// TIA Portal project "BHX_PLC_2_V17" (V17)

(* hardware
DEVICE "ET 200SP station_1"  ET 200SP-Station
   slot 0: "Rack_0"  Rack  6ES5 710-8MAx1
   slot 1: "k1bhx01cpu"  CPU 1510SP-1 PN  6ES7 510-1DJ01-0AB0  V2.8
      slot 32768: "PROFINET interface_1"  X1
         slot 32771: "Port_3"  X1 P3
   slot 2: "DI 8x24VDC BA_1"  DI 8x24VDC BA  6ES7 131-6BF01-0AA0  V0.0
      slot 1: "DI 8x24VDC BA_1"  DI 8x24VDC BA
   slot 3: "DI 8x24VDC BA_2"  DI 8x24VDC BA  6ES7 131-6BF01-0AA0  V0.0
      slot 1: "DI 8x24VDC BA_2"  DI 8x24VDC BA
   slot 4: "DQ 8x24VDC/0.5A ST_1"  DQ 8x24VDC/0.5A ST  6ES7 132-6BF01-0BA0  V0.0
      slot 1: "DQ 8x24VDC/0.5A ST_1"  DQ 8x24VDC/0.5A ST
   slot 5: "Server module_1"  Server module  6ES7 193-6PA00-0AA0  V1.1
      slot 1: "Server module_1"  Server module
   slot 127: "BA 2xRJ45"  BA 2xRJ45  6ES7 193-6AR00-0AA0  V0.0
      slot 32769: "Port_1"  X1 P1  6ES7 193-6AR00-0AA0
      slot 32770: "Port_2"  X1 P2  6ES7 193-6AR00-0AA0
DEVICE "ET 200SP station_2"  ET 200SP-Station
   slot 0: "Rack_0"  Rack  6ES5 710-8MAx1
   slot 0: "et-bhx"  IM 155-6 PN ST  6ES7 155-6AU01-0BN0  V4.1
   slot 1: "DI 8x24VDC BA_1"  DI 8x24VDC BA  6ES7 131-6BF01-0AA0  V0.0
      slot 1: "DI 8x24VDC BA_1"  DI 8x24VDC BA
   slot 2: "DQ 8x24VDC/0.5A ST_1"  DQ 8x24VDC/0.5A ST  6ES7 132-6BF01-0BA0  V0.0
      slot 1: "DQ 8x24VDC/0.5A ST_1"  DQ 8x24VDC/0.5A ST
   slot 3: "AI 4xU/I 2-wire ST_1"  AI 4xU/I 2-wire ST  6ES7 134-6HD01-0BA1  V2.0
      slot 1: "AI 4xU/I 2-wire ST_1"  AI 4xU/I 2-wire ST
   slot 4: "Server module_1"  Server module  6ES7 193-6PA00-0AA0  V1.1
      slot 1: "Server module_1"  Server module
   slot 127: "BA 2xRJ45"  BA 2xRJ45  6ES7 193-6AR00-0AA0  V0.0
      slot 1: "Port_1"  X1 P1 R  6ES7 193-6AR00-0AA0  V0.0
      slot 2: "Port_2"  X1 P2 R  6ES7 193-6AR00-0AA0  V0.0
DEVICE "GSD device_1"  GSD.Device.PN
   slot 0: "Rack"  Rack  V1.0
   slot 0: "k1bhx011"  KRC4-ProfiNet_4.1  0x300  V4.1
      slot 0: "KRC4-ProfiNet_4.1"  KRC4-ProfiNet_4.1
      slot 1: "Interface1"  Interface1
         slot 1: "Port1"  Port1
   slot 2: "1024 digital in- and outputs_1"  1024 digital in- and outputs  KUKA Device IO1024
      slot 0: "1024 digital in- and outputs"  1024 digital in- and outputs
DEVICE "GSD device_2"  GSD.Device.PN
   slot 0: "Rack"  Rack  V1.0
   slot 0: "matrixbhx"  Matrix 320  M320  V1.37.0
      slot 0: "Matrix 320"  Matrix 320
      slot 1: "1 Port PN-RT"  1 Port PN-RT
         slot 1: "Port 1"  Port 1
   slot 1: "Virtual 8 Byte Output"  Virtual 8 Byte Output
      slot 0: "Virtual 8 Byte Output"  Virtual 8 Byte Output
   slot 2: "Virtual 64 Byte Input"  Virtual 64 Byte Input
      slot 0: "Virtual 64 Byte Input"  Virtual 64 Byte Input
*)

// ===== PLC "k1bhx01cpu"  CPU 1510SP-1 PN =====

VAR_GLOBAL   // PLC tag table "PLC_Machine_IO"
   "PLC_WorkpieceAtStopper" AT %Q0.0 : Bool;
   "PLC_InfeedAreaFree" AT %Q0.1 : Bool;
   "PLC_OutfeedAreaFree" AT %Q0.2 : Bool;
   "PLC_OpenClamps" AT %Q0.3 : Bool;
   "PLC_ResetMcc" AT %Q0.4 : Bool;
   "PLC_InfeedPositionFree" AT %I0.0 : Bool;
   "PLC_WorkpieceClamped" AT %I0.1 : Bool;
   "PLC_WorkpieceRdyToTurn" AT %I0.2 : Bool;
   "PLC_WorkpiecePickupPos1" AT %I0.3 : Bool;
   "PLC_WorkpiecePickupPos2" AT %I0.4 : Bool;
   "PLC_AutoFeedingModeActive" AT %I0.5 : Bool;
   "PLC_StopperWorkpos" AT %I0.6 : Bool;
END_VAR

VAR_GLOBAL   // PLC tag table "Robot_Machine_IO"
   "WorkpieceAtStopper" AT %I20.0 : Bool;
   "InfeedAreaFree" AT %I20.1 : Bool;
   "OutfeedAreaFree" AT %I20.2 : Bool;
   "OpenClamps" AT %I20.3 : Bool;
   "ResetMcc" AT %I20.4 : Bool;
   "InfeedPositionFree" AT %Q20.0 : Bool;
   "WorkpieceClamped" AT %Q20.1 : Bool;
   "WorkpieceRdyToTurn" AT %Q20.2 : Bool;
   "WorkpiecePickupPos1" AT %Q20.3 : Bool;
   "WorkpiecePickupPos2" AT %Q20.4 : Bool;
   "AutoFeedingModeActive" AT %Q20.5 : Bool;
   "StopperWorkpos" AT %Q20.6 : Bool;
END_VAR

VAR_GLOBAL   // PLC tag table "ET200_Gripper"
   "InGripperMainHome1" AT %I10.0 : Bool;
   "InGripperRetracted" AT %I10.1 : Bool;
   "InGripperMainHome2" AT %I10.2 : Bool;
   "InGripperFeederHome" AT %I10.3 : Bool;
   "OutVacuumON" AT %Q10.0 : Bool;
   "InGripperGerconNC" AT %I10.4 : Bool;
   "InGripperVacuumNC" AT %I10.5 : Bool;
   "InGripperRangefinder" AT %IW14 : Int;
   "OutPressureOFF" AT %Q10.1 : Bool;
   "OutGripperMainRetract" AT %Q10.2 : Bool;
   "OutFlow2Part" AT %Q10.3 : Bool;
END_VAR

VAR_GLOBAL   // PLC tag table "KUKA_To_PLC"
   "From_KUKA_ALARM_STOP_KRC" AT %I35.1 : Bool;   // KUKA. Аварийный СТОП (122)
   "From_KUKA_EXT_ACTIVE" AT %I35.7 : Bool;   // KUKA. В режиме Внешняя Автоматика (128)
   "From_KUKA_PERI_RDY_KRC" AT %I35.5 : Bool;   // KUKA. Готовность приводов (126)
   "From_KUKA_STOPMESS_KRC" AT %I35.3 : Bool;   // KUKA. СТОП (124)
   "From_KUKA_IN_HOME_KRC" AT %I36.0 : Bool;   // KUKA. В домашней позиции (129)
   "From_KUKA_PRO_MOVE_KRC" AT %I36.7 : Bool;   // KUKA. Робот в движении (136)
   "From_KUKA_PGNO_REFL_KRC" AT %IW37 : UInt;   // KUKA. Активный номер программы (137-152)
   "From_KUKA_PGNO_REQ_KRC" AT %I36.2 : Bool;   // KUKA. Запрос на новую программу (131)
   "From_KUKA_USER_SAF_KRC" AT %I35.4 : Bool;   // KUKA. Безопасность оператора (125)
   "From_KUKA_ROB_CAL_KRC" AT %I36.1 : Bool;   // KUKA. Юстировка выполнена (130)
   "From_KUKA_I_O_ACTCONF_KRC" AT %I35.2 : Bool;   // KUKA. Внешняя автоматика сконфигурирована (123)
   "From_KUKA_RC_RDY1_KRC" AT %I35.0 : Bool;   // KUKA. Готовность приводов (121)
   "From_KUKA_APPL_RUN_KRC" AT %I36.3 : Bool;   // KUKA. Приложение запущено (132)
   "From_KUKA_Cam" AT %I21.3 : Bool;   // KUKA. Запрос на сканирование (12)
   "From_KUKA_LifeBit" AT %I35.6 : Bool;   // KUKA. Бит Жизни (127)
   "From_KUKA_EXT_FIRST_START" AT %I36.5 : Bool;   // KUKA. Начальный запуск внешней автоматики (134)
   "From_KUKA_SetVacuumON" AT %I21.0 : Bool;   // KUKA. Включить вакуум (9)
   "From_KUKA_SetPressureOFF" AT %I21.1 : Bool;   // KUKA. Выключить давление (10)
   "From_KUKA_SetRetract" AT %I21.2 : Bool;   // KUKA. Задвинуть цилиндры (11)
   "From_KUKA_Flow2PartON" AT %I21.5 : Bool;   // KUKA. Включить поддув деталей (14)
   "From_KUKA_SetFlipClose" AT %I21.4 : Bool;   // KUKA. Закрыть стол переворота(13)
   "From_KUKA_PartOK" AT %I22.0 : Bool;   // KUKA. Деталь ОК (17)
   "From_KUKA_PartMeasuring" AT %I21.7 : Bool;   // KUKA. Измерение детали (16)
   "From_KUKA_PRO_ACT_KRC" AT %I36.6 : Bool;   // KUKA. Программа активна (135)
   "From_KUKA_ERROR_KRC" AT %I36.4 : Bool;   // KUKA. Ошибка на роботе (133)
   "From_KUKA_AXIS_ACT_A1" AT %IW24 : UInt;   // KUKA. Угол поворота оси А1 робота плюс 180 градусов (33-48)
   "From_KUKA_POS_ACT_Z" AT %IW30 : UInt;   // KUKA. Координата Z актуальной позиции робота (81-96)
   "From_KUKA_POS_ACT_Y" AT %IW28 : UInt;   // KUKA. Координата Y актуальной позиции робота (65-80)
   "From_KUKA_POS_ACT_X" AT %IW26 : UInt;   // KUKA. Координата X актуальной позиции робота (49-64)
   "From_KUKA_POS_ACT_A" AT %IW32 : UInt;   // KUKA. Угол A актуальной позиции робота (97-112)
   "From_KUKA_Pallet_Scanned" AT %I39.0 : Bool;   // KUKA. Робот в движении (153)
   "From_KUKA_FlipVacuumOn" AT %I21.6 : Bool;   // KUKA. Включить вакуум стола (15)
   "From_KUKA_Part_Status" AT %IW40 : UInt;   // KUKA. Статус детали (161-176)
   "From_KUKA_Serial_Number" AT %IW42 : UInt;   // KUKA. Серийный номер (177-192)
END_VAR

VAR_GLOBAL   // PLC tag table "PLC_To_KUKA"
   "To_KUKA_Rangefinder" AT %QW43 : UInt;   // PLC. Дальномер (185-200)
   "To_KUKA_Gercon" AT %Q21.4 : Bool;   // PLC. Касание листа нормальное (13)
   "To_KUKA_PLC_STOP" AT %Q32.3 : Bool;   // PLC. ПЛК - СТОП (100)
   "To_KUKA_PAUSE_STOP" AT %Q32.4 : Bool;   // PLC. ПЛК - ПАУЗА (101)
   "To_KUKA_MOVE_ENABLE_KRC" AT %Q35.1 : Bool;   // PLC. Разрешение на перемещение (122)
   "To_KUKA_PGNO_KRC" AT %QW33 : UInt;   // PLC. Номер программы (105-120)
   "To_KUKA_PGNO_VALID_KRC" AT %Q35.6 : Bool;   // PLC. Корректность номера программы 127
   "To_KUKA_PGNO_PARITY" AT %Q35.5 : Bool;   // PLC. Чётность номера программы 126
   "To_KUKA_CONF_MESS" AT %Q35.2 : Bool;   // PLC. Подтверждение сообщения 123
   "To_KUKA_DRIVERS_OFF" AT %Q35.4 : Bool;   // PLC. Отключить привода 125
   "To_KUKA_DRIVERS_ON" AT %Q35.3 : Bool;   // PLC. Включить привода 124
   "To_KUKA_Collision" AT %Q21.5 : Bool;   // PLC. Касание аварийное (14)
   "To_KUKA_QRcode_X" AT %QW37 : UInt;   // PLC. Отклонение по оси X (137-152)
   "To_KUKA_QRcode_Angle" AT %QW41 : UInt;   // PLC. Отклонение по углу (169-184)
   "To_KUKA_EXT_START_KRC" AT %Q35.0 : Bool;   // PLC. Внешний страт (121)
   "To_KUKA_Vacuum_Ok" AT %Q21.6 : Bool;   // PLC. Вакуум ОК (15)
   "To_KUKA_QRcode_Y" AT %QW39 : UInt;   // PLC. Отклонение по оси Y (153-168)
   "To_KUKA_Cam_Ok" AT %Q21.7 : Bool;   // PLC. Камера ОК (16)
   "To_KUKA_IsGripperMainHome" AT %Q21.0 : Bool;   // PLC. Геркон основного цилиндра (9)
   "To_KUKA_IsGripperFeederHome" AT %Q21.1 : Bool;   // PLC. Геркон цилиндра подачи (10)
   "To_KUKA_Part_length_X" AT %QW45 : UInt;   // PLC. Длинна детали по X (201-216)
   "To_KUKA_Part_thickness_Z" AT %QW49 : UInt;   // PLC. Ширина детали по Z (233-248)
   "To_KUKA_GripperRetracted" AT %Q22.0 : Bool;   // PLC. Концевой выключатель (17)
   "To_KUKA_PartEndSwitch_1" AT %Q22.1 : Bool;   // PLC. Концевой выключатель (18)
   "To_KUKA_PartEndSwitch_2" AT %Q22.2 : Bool;   // PLC. Концевой выключатель (19)
   "To_KUKA_Gripper_Sign_X" AT %Q22.3 : Bool;   // PLC. Сдвиг захвата по X (20)
   "To_KUKA_Gripper_Sign_Y" AT %Q22.4 : Bool;   // PLC. Сдвиг захвата по Y (21)
   "To_KUKA_FlipTableOpened" AT %Q22.6 : Bool;   // PLC. Стол для переворота открыт (23)
   "To_KUKA_FlipTableClosed" AT %Q22.7 : Bool;   // PLC. Стол для переворота закрыт (24)
   "To_KUKA_Part_length_Y" AT %QW47 : UInt;   // PLC. Длинна детали по Y (217-232)
   "To_KUKA_QRcode_Z" AT %QW51 : UInt;   // PLC. Отклонение по высоте (249-264)
   "To_KUKA_Part_X" AT %QW53 : UInt;   // PLC. Отклонение по оси X (265-280)
   "To_KUKA_Part_Y" AT %QW55 : UInt;   // PLC. Отклонение по оси Y (281-296)
   "To_KUKA_Part_A" AT %QW59 : UInt;   // PLC. Отклонение по углу (313-328)
   "To_KUKA_Part_Z" AT %QW57 : UInt;   // PLC. Отклонение по высоте (297-312)
   "To_KUKA_Part_Length_X0" AT %QW61 : UInt;   // PLC. Отклонение по высоте (329-344)
   "To_KUKA_Part_Length_Y0" AT %QW63 : UInt;   // PLC. Отклонение по углу (345-360)
   "To_KUKA_Gripper_Within_part" AT %Q22.5 : Bool;   // PLC. Захват соприкасается с деталью полностью (22)
   "To_KUKA_Part_Slot" AT %QW65 : UInt;   // PLC. Отклонение по углу (361-376)
   "To_KUKA_Free_Slot" AT %QW67 : UInt;   // PLC. Отклонение по углу (377-392)
   "To_KUKA_AckPalletScanned" AT %Q32.5 : Bool;   // PLC. Подтверждение сканирования поддона 102
   "To_KUKA_Slot_X" AT %QW69 : UInt;   // PLC. Отклонение по оси X (393-408)
   "To_KUKA_Slot_Y" AT %QW71 : UInt;   // PLC. Отклонение по оси Y (409-424)
   "To_KUKA_Slot_Z" AT %QW73 : UInt;   // PLC. Отклонение по высоте (425-440)
   "To_KUKA_Slot_A" AT %QW75 : UInt;   // PLC. Отклонение по углу (441-456)
   "To_KUKA_WithoutMachine" AT %Q32.6 : Bool;   // PLC. Работа без машины 103
   "To_KUKA_Part_Destination" AT %QW77 : UInt;   // PLC. Назначение детали (457-472)
   "To_KUKA_Out_X" AT %QW79 : UInt;   // PLC. Отклонение по оси X (473-488)
   "To_KUKA_Out_Y" AT %QW81 : UInt;   // PLC. Отклонение по оси Y (489-544)
   "To_KUKA_Out_Z" AT %QW83 : UInt;   // PLC. Отклонение по высоте (505-520)
   "To_KUKA_Out_A" AT %QW85 : UInt;   // PLC. Отклонение по углу (521-536)
END_VAR

VAR_GLOBAL   // PLC tag table "Matrix"
   "MatrixPhase_ON" AT %Q148.7 : Bool;
   "MatrixGoobRead" AT %I148.0 : Bool;
   "MatrixBadRead" AT %I148.1 : Bool;
END_VAR

VAR_GLOBAL   // PLC tag table "Operator_panel"
   "button_Alarm" AT %I1.0 : Bool;
   "button_Pause" AT %I1.1 : Bool;
   "button_Reset" AT %I1.2 : Bool;
   "button_Start" AT %I1.3 : Bool;
END_VAR

VAR_GLOBAL   // PLC tag table "FlipTable"
   "OutFlipClose" AT %Q0.5 : Bool;
   "OutFlipVacuumOn" AT %Q0.6 : Bool;
END_VAR

VAR_GLOBAL   // PLC tag table "RobotTask"
   "task_status" AT %Q1000.0 : "Char_30";
   "part_status" AT %Q1030.0 : "Char_30";
END_VAR

VAR_GLOBAL   // PLC tag table "PLC_To_VC"
   "To_VC_Rangefinder" AT %QW343 : UInt;   // PLC. Дальномер (185-200)
   "To_VC_Gercon" AT %Q321.4 : Bool;   // PLC. Касание листа нормальное (13)
   "To_VC_PLC_STOP" AT %Q332.3 : Bool;   // PLC. ПЛК - СТОП (100)
   "To_VC_PAUSE_STOP" AT %Q332.4 : Bool;   // PLC. ПЛК - ПАУЗА (101)
   "To_VC_MOVE_ENABLE_KRC" AT %Q335.1 : Bool;   // PLC. Разрешение на перемещение (122)
   "To_VC_PGNO_KRC" AT %QW333 : UInt;   // PLC. Номер программы (105-120)
   "To_VC_PGNO_VALID_KRC" AT %Q335.6 : Bool;   // PLC. Корректность номера программы 127
   "To_VC_PGNO_PARITY" AT %Q335.5 : Bool;   // PLC. Чётность номера программы 126
   "To_VC_CONF_MESS" AT %Q335.2 : Bool;   // PLC. Подтверждение сообщения 123
   "To_VC_DRIVERS_OFF" AT %Q335.4 : Bool;   // PLC. Отключить привода 125
   "To_VC_DRIVERS_ON" AT %Q335.3 : Bool;   // PLC. Включить привода 124
   "To_VC_Collision" AT %Q321.5 : Bool;   // PLC. Касание аварийное (14)
   "To_VC_QRcode_X" AT %QW337 : UInt;   // PLC. Отклонение по оси X (137-152)
   "To_VC_QRcode_Angle" AT %QW341 : UInt;   // PLC. Отклонение по углу (169-184)
   "To_VC_EXT_START_KRC" AT %Q335.0 : Bool;   // PLC. Внешний страт (121)
   "To_VC_Vacuum_Ok" AT %Q321.6 : Bool;   // PLC. Вакуум ОК (15)
   "To_VC_QRcode_Y" AT %QW339 : UInt;   // PLC. Отклонение по оси Y (153-168)
   "To_VC_Cam_Ok" AT %Q321.7 : Bool;   // PLC. Камера ОК (16)
   "To_VC_IsGripperMainHome" AT %Q321.0 : Bool;   // PLC. Геркон основного цилиндра (9)
   "To_VC_IsGripperFeederHome" AT %Q321.1 : Bool;   // PLC. Геркон цилиндра подачи (10)
   "To_VC_Part_length_X" AT %QW345 : UInt;   // PLC. Длинна детали по X (201-216)
   "To_VC_Part_thickness_Z" AT %QW349 : UInt;   // PLC. Ширина детали по Z (233-248)
   "To_VC_GripperRetracted" AT %Q322.0 : Bool;   // PLC. Концевой выключатель (17)
   "To_VC_PartEndSwitch_1" AT %Q322.1 : Bool;   // PLC. Концевой выключатель (18)
   "To_VC_PartEndSwitch_2" AT %Q322.2 : Bool;   // PLC. Концевой выключатель (19)
   "To_VC_Gripper_Sign_X" AT %Q322.3 : Bool;   // PLC. Сдвиг захвата по X (20)
   "To_VC_Gripper_Sign_Y" AT %Q322.4 : Bool;   // PLC. Сдвиг захвата по Y (21)
   "To_VC_FlipTableOpened" AT %Q322.6 : Bool;   // PLC. Стол для переворота открыт (23)
   "To_VC_FlipTableClosed" AT %Q322.7 : Bool;   // PLC. Стол для переворота закрыт (24)
   "To_VC_Part_length_Y" AT %QW347 : UInt;   // PLC. Длинна детали по Y (217-232)
   "To_VC_QRcode_Z" AT %QW351 : UInt;   // PLC. Отклонение по высоте (249-264)
   "To_VC_Part_X" AT %QW353 : UInt;   // PLC. Отклонение по оси X (265-280)
   "To_VC_Part_Y" AT %QW355 : UInt;   // PLC. Отклонение по оси Y (281-296)
   "To_VC_Part_A" AT %QW359 : UInt;   // PLC. Отклонение по углу (313-328)
   "To_VC_Part_Z" AT %QW357 : UInt;   // PLC. Отклонение по высоте (297-312)
   "To_VC_Part_Length_X0" AT %QW361 : UInt;   // PLC. Отклонение по высоте (329-344)
   "To_VC_Part_Length_Y0" AT %QW363 : UInt;   // PLC. Отклонение по углу (345-360)
   "To_VC_Gripper_Within_part" AT %Q322.5 : Bool;   // PLC. Захват соприкасается с деталью полностью (22)
   "To_VC_Part_Slot" AT %QW365 : UInt;   // PLC. Отклонение по углу (361-376)
   "To_VC_Free_Slot" AT %QW367 : UInt;   // PLC. Отклонение по углу (377-392)
   "To_VC_AckPalletScanned" AT %Q332.5 : Bool;   // PLC. Подтверждение сканирования поддона 102
   "To_VC_Slot_X" AT %QW369 : UInt;   // PLC. Отклонение по оси X (393-408)
   "To_VC_Slot_Y" AT %QW371 : UInt;   // PLC. Отклонение по оси Y (409-424)
   "To_VC_Slot_Z" AT %QW373 : UInt;   // PLC. Отклонение по высоте (425-440)
   "To_VC_Slot_A" AT %QW375 : UInt;   // PLC. Отклонение по углу (441-456)
   "To_VC_WithoutMachine" AT %Q332.6 : Bool;   // PLC. Работа без машины 103
   "To_VC_Part_Destination" AT %QW377 : UInt;   // PLC. Назначение детали (457-472)
   "To_VC_Out_X" AT %QW379 : UInt;   // PLC. Отклонение по оси X (473-488)
   "To_VC_Out_Y" AT %QW381 : UInt;   // PLC. Отклонение по оси Y (489-544)
   "To_VC_Out_Z" AT %QW383 : UInt;   // PLC. Отклонение по высоте (505-520)
   "To_VC_Out_A" AT %QW385 : UInt;   // PLC. Отклонение по углу (521-536)
   "To_VC_Test_DInt" AT %QD388 : DInt;   // PLC. Tecт
END_VAR

VAR_GLOBAL   // PLC tag table "VC_To_PLC"
   "From_VC_ALARM_STOP_KRC" AT %I335.1 : Bool;   // KUKA. Аварийный СТОП (122)
   "From_VC_EXT_ACTIVE" AT %I335.7 : Bool;   // KUKA. В режиме Внешняя Автоматика (128)
   "From_VC_PERI_RDY_KRC" AT %I335.5 : Bool;   // KUKA. Готовность приводов (126)
   "From_VC_STOPMESS_KRC" AT %I335.3 : Bool;   // KUKA. СТОП (124)
   "From_VC_IN_HOME_KRC" AT %I336.0 : Bool;   // KUKA. В домашней позиции (129)
   "From_VC_PRO_MOVE_KRC" AT %I336.7 : Bool;   // KUKA. Робот в движении (136)
   "From_VC_PGNO_REFL_KRC" AT %IW337 : UInt;   // KUKA. Активный номер программы (137-152)
   "From_VC_PGNO_REQ_KRC" AT %I336.2 : Bool;   // KUKA. Запрос на новую программу (131)
   "From_VC_USER_SAF_KRC" AT %I335.4 : Bool;   // KUKA. Безопасность оператора (125)
   "From_VC_ROB_CAL_KRC" AT %I336.1 : Bool;   // KUKA. Юстировка выполнена (130)
   "From_VC_I_O_ACTCONF_KRC" AT %I335.2 : Bool;   // KUKA. Внешняя автоматика сконфигурирована (123)
   "From_VC_RC_RDY1_KRC" AT %I335.0 : Bool;   // KUKA. Готовность приводов (121)
   "From_VC_APPL_RUN_KRC" AT %I336.3 : Bool;   // KUKA. Приложение запущено (132)
   "From_VC_Cam" AT %I321.3 : Bool;   // KUKA. Запрос на сканирование (12)
   "From_VC_LifeBit" AT %I335.6 : Bool;   // KUKA. Бит Жизни (127)
   "From_VC_EXT_FIRST_START" AT %I336.5 : Bool;   // KUKA. Начальный запуск внешней автоматики (134)
   "From_VC_SetVacuumON" AT %I321.0 : Bool;   // KUKA. Включить вакуум (9)
   "From_VC_SetPressureOFF" AT %I321.1 : Bool;   // KUKA. Выключить давление (10)
   "From_VC_SetRetract" AT %I321.2 : Bool;   // KUKA. Задвинуть цилиндры (11)
   "From_VC_Flow2PartON" AT %I321.5 : Bool;   // KUKA. Включить поддув деталей (14)
   "From_VC_SetFlipClose" AT %I321.4 : Bool;   // KUKA. Закрыть стол переворота(13)
   "From_VC_PartOK" AT %I322.0 : Bool;   // KUKA. Деталь ОК (17)
   "From_VC_PartMeasuring" AT %I321.7 : Bool;   // KUKA. Измерение детали (16)
   "From_VC_PRO_ACT_KRC" AT %I336.6 : Bool;   // KUKA. Программа активна (135)
   "From_VC_ERROR_KRC" AT %I336.4 : Bool;   // KUKA. Ошибка на роботе (133)
   "From_VC_AXIS_ACT_A1" AT %IW324 : UInt;   // KUKA. Угол поворота оси А1 робота плюс 180 градусов (33-48)
   "From_VC_POS_ACT_Z" AT %IW330 : UInt;   // KUKA. Координата Z актуальной позиции робота (81-96)
   "From_VC_POS_ACT_Y" AT %IW328 : UInt;   // KUKA. Координата Y актуальной позиции робота (65-80)
   "From_VC_POS_ACT_X" AT %IW326 : UInt;   // KUKA. Координата X актуальной позиции робота (49-64)
   "From_VC_POS_ACT_A" AT %IW332 : UInt;   // KUKA. Угол A актуальной позиции робота (97-112)
   "From_VC_Pallet_Scanned" AT %I339.0 : Bool;   // KUKA. Робот в движении (153)
   "From_VC_FlipVacuumOn" AT %I321.6 : Bool;   // KUKA. Включить вакуум стола (15)
   "From_VC_Part_Status" AT %IW340 : UInt;   // KUKA. Статус детали (161-176)
   "From_VC_Serial_Number" AT %IW342 : UInt;   // KUKA. Серийный номер (177-192)
END_VAR

TYPE "PLC_Tag"
   STRUCT
      "Name" : String[30];
      "Type" : String[30];
      Use : String[5];
      ReadOnly : USInt;
      DB_number : UInt;
      OffsetByte : UInt;
      OffsetBit : USInt;
      Robot_number : USInt;
   END_STRUCT;
END_TYPE

TYPE "InStatus"
   STRUCT
      previous_programs : Array[1..5] of Int;
      machine_status : String[30];
      robot_status : String[30];
      part_status : String[30];
      operation_types : Array[1..5] of String[30];
      lay_number : Int := -1;
      operation_side : String[4];
      part_side : String[4];
   END_STRUCT;
   // previous_programs[1] := -1;
   // previous_programs[2] := -1;
   // previous_programs[3] := -1;
   // previous_programs[4] := -1;
   // previous_programs[5] := -1;
END_TYPE

TYPE "RobotProgram"
   STRUCT
      trajectory : String[30];
      Entry_Points : Array[1..12] of "EntryPoint";
      OUT_Status : "OutStatus";
   END_STRUCT;
END_TYPE

TYPE "OutStatus"
   STRUCT
      inprocess_task_status : String[30];
      inprocess_part_status : String[30];
      finish_task_status : String[30];
      finish_part_status : String[30];
   END_STRUCT;
END_TYPE

TYPE "EntryPoint"
   STRUCT
      active : Bool;
      previous_trajectory : String[30];
      machine_status : String[30];
      robot_status : String[30];
      part_status : String[30];
      part_destination : String[30];
      operation_type : String[30];
      lay_number : Int := -1;
      operation_side : String[1] := '';
      part_side : String[1] := '';
   END_STRUCT;
END_TYPE

TYPE "TypeRobotTask"
   STRUCT
      not_sended2Arduino : Bool;
      not_sended2BHX : Bool;
      new_part : Bool;
      start_job : Bool;
      reset_job : Bool;
      robot_alarm_reset : Bool;
      "w/o_machine_mode" : Bool;
      gripper_sign_X : Bool;
      gripper_sign_Y : Bool;
      gripper_within_part : Bool;
      robot_pause : Bool;
      pallet_scanned : Bool;
      new_pallet : Bool;
      robot_in_home : Bool;
      program_fullpath : String[99];
      part_length_X : UInt;
      part_length_Y : UInt;
      part_thickness_Z : UInt;
      part_pos_X : Real;
      part_pos_Y : Real;
      part_pos_Z : Real;
      part_angle_A : Real;
      part_side : Char;
      part_slot : USInt;
      free_slot : USInt;
      operation_side : Char;
      operation_number : Int;
      lay_number : Int;
      robot_task_id : LInt;
      robot_id : LInt;
      part_id : LInt;
      part_number : LInt;
      order_id : LInt;
      plc_id : LInt;
      robot_program : UInt;
      operation_type : String[30];
      machine_status : String[30];
      robot_trajectory : String[30];
      robot_status : String[30];
      task_status : String[30];
      part_status : String[30];
      part_source : String[30];
      part_destination : String[30];
      plc_ip : String[30];
      plc_name : String[30];
      robot_name : String[30];
      part_length_X0 : UInt;
      part_length_Y0 : UInt;
      slot_pos_X : Real;
      slot_pos_Y : Real;
      slot_pos_Z : Real;
      slot_angle_A : Real;
      out_pos_X : Real;
      out_pos_Y : Real;
      out_pos_Z : Real;
      out_pos_A : Real;
      robot_serial : UInt;
      Test_DInt : DInt;
   END_STRUCT;
END_TYPE

TYPE "Char_30"
   STRUCT
      str : Array[1..30] of Char;
   END_STRUCT;
END_TYPE

TYPE "TypeRobotTaskChar"
   STRUCT
      not_sended2Arduino : Bool;
      not_sended2BHX : Bool;
      new_part : Bool;
      start_job : Bool;
      reset_job : Bool;
      robot_alarm_reset : Bool;
      "w/o_machine_mode" : Bool;
      gripper_sign_X : Bool;
      gripper_sign_Y : Bool;
      gripper_within_part : Bool;
      robot_pause : Bool;
      pallet_scanned : Bool;
      new_pallet : Bool;
      robot_in_home : Bool;
      program_fullpath : "Char_99";
      part_length_X : UInt;
      part_length_Y : UInt;
      part_thickness_Z : UInt;
      part_pos_X : Real;
      part_pos_Y : Real;
      part_pos_Z : Real;
      part_angle_A : Real;
      part_side : Char;
      part_slot : USInt;
      free_slot : USInt;
      operation_side : Char;
      operation_number : Int;
      lay_number : Int;
      robot_task_id : LInt;
      robot_id : LInt;
      part_id : LInt;
      part_number : LInt;
      order_id : LInt;
      plc_id : LInt;
      robot_program : UInt;
      operation_type : "Char_30";
      machine_status : "Char_30";
      robot_trajectory : "Char_30";
      robot_status : "Char_30";
      task_status : "Char_30";
      part_status : "Char_30";
      part_source : "Char_30";
      part_destination : "Char_30";
      plc_ip : "Char_30";
      plc_name : "Char_30";
      robot_name : "Char_30";
      part_length_X0 : UInt;
      part_length_Y0 : UInt;
      slot_pos_X : Real;
      slot_pos_Y : Real;
      slot_pos_Z : Real;
      slot_angle_A : Real;
   END_STRUCT;
END_TYPE

TYPE "Char_99"
   STRUCT
      str : Array[1..99] of Char;
   END_STRUCT;
END_TYPE

TYPE "Alarm"
   STRUCT
      bGenAlarm : Bool;   // Авария
      bGenWarning : Bool;   // Предупреждения
      bAlarmReset : Bool;   // Сброс
      A_bAlarmButtonPushed : Bool;   // Аварийная кнопка
      A_bPressureLoss : Bool;   // Авария. Низкое давление
      A_bCantContinueTask : Bool;   // Авария. Не может продолжать задание
      W_bRobotSubmitDown : Bool;   // Робот. Бит жизни
      W_bRobotStop : Bool;   // Робот. Аварийный останов
      W_bRobotUserSafe : Bool;   // Робот. Защита пользователя
      W_bGripperTooDown : Bool;   // Захват. Ниже допустимой точки
      W_bGripperSheetLost : Bool;   // Захват. Ошибка взятия листа
      W_bGripperSheetTakeFail : Bool;   // Захват. Листа не оказалось на посту
      W_bCameraCantFind : Bool;   // Камера. Ошибка захвата изображения
      bSTOP : Bool;   // СТОП
      bPAUSE : Bool;   // ПАУЗА
   END_STRUCT;
END_TYPE

DATA_BLOCK "Default_SupervisionDB"   // DB13
{ S7_Optimized_Access := 'TRUE' }
VERSION : 0.1
// stored: InstanceOfName Default_SupervisionFB
"Default_SupervisionFB"
BEGIN
END_DATA_BLOCK

// folder: 1_Alerts

DATA_BLOCK "Driver_Alerts_DB"   // DB4
{ S7_Optimized_Access := 'TRUE' }
VERSION : 0.1
// stored: InstanceOfName Driver_Alerts
"Driver_Alerts"
BEGIN
END_DATA_BLOCK

// folder: 2_Robot

DATA_BLOCK "Get_Robot_Program_DB"   // DB8
{ S7_Optimized_Access := 'TRUE' }
VERSION : 0.1
   VAR
      i : UInt;
      j : UInt;
      operation_type_ok : Bool;
      machine_status_ok : Bool;
      robot_status_ok : Bool;
      part_status_ok : Bool;
      first_program_ok : Bool;
      previous_trajectory_ok : Bool;
      program_ok : Bool;
      lay_ok : Bool;
      operation_side_ok : Bool;
      part_side_ok : Bool;
      part_destination_ok : Bool;
      entryPoint_active : Bool;
   END_VAR
BEGIN
END_DATA_BLOCK

// folder: 2_Robot/DB

DATA_BLOCK "KUKA_Data"   // DB2
{ S7_Optimized_Access := 'TRUE' }
VERSION : 0.1
   VAR
      PGNO_REFL_KRC : Int;   // KUKA. Активный номер программы (41-56)
      PGNO_KRC : Int;   // PLC. Номер программы (73-88)
   END_VAR
BEGIN
END_DATA_BLOCK

DATA_BLOCK "!Robot_DB"   // DB3
{ S7_Optimized_Access := 'TRUE' }
VERSION : 0.1
// stored: InstanceOfName !Robot
"!Robot"
BEGIN
END_DATA_BLOCK

DATA_BLOCK "KUKA_IO_DB"   // DB7
{ S7_Optimized_Access := 'TRUE' }
VERSION : 0.1
// stored: InstanceOfName KUKA_IO
"KUKA_IO"
BEGIN
END_DATA_BLOCK

DATA_BLOCK "RobotExternalStart"   // DB211
{ S7_Optimized_Access := 'TRUE' }
VERSION : 0.1
// stored: InstanceOfName Driver_RobotExternalStart
"Driver_RobotExternalStart"
BEGIN
END_DATA_BLOCK

DATA_BLOCK "RobotPause_DB"   // DB212
{ S7_Optimized_Access := 'TRUE' }
VERSION : 0.1
// stored: InstanceOfName Driver_RobotPause
"Driver_RobotPause"
BEGIN
END_DATA_BLOCK

DATA_BLOCK "Alerts_DB"   // DB511
{ S7_Optimized_Access := 'TRUE' }
VERSION : 0.1
// stored: InstanceOfName Driver_Alerts
"Driver_Alerts"
BEGIN
END_DATA_BLOCK

// folder: 3_Gripper

DATA_BLOCK "Driver_Gripper_DB"   // DB31
{ S7_Optimized_Access := 'TRUE' }
VERSION : 0.1
// stored: InstanceOfName Driver_Gripper
"Driver_Gripper"
BEGIN
END_DATA_BLOCK

DATA_BLOCK "!Gripper_DB"   // DB300
{ S7_Optimized_Access := 'TRUE' }
VERSION : 0.1
// stored: InstanceOfName Driver_Gripper
"Driver_Gripper"
BEGIN
END_DATA_BLOCK

// folder: 4_Working

DATA_BLOCK "Working_DB"   // DB15
{ S7_Optimized_Access := 'TRUE' }
VERSION : 0.1
// stored: InstanceOfName Driver_Working
"Driver_Working"
BEGIN
END_DATA_BLOCK

DATA_BLOCK "Robot_Programs"   // DB23
{ S7_Optimized_Access := 'FALSE' }
VERSION : 0.1
   VAR
      Count : USInt := 18;
      List : Array[0..21] of "RobotProgram";
   END_VAR
BEGIN
   List[4].Entry_Points[7].part_side := '';
   List[4].Entry_Points[7].operation_side := '';
   List[4].Entry_Points[7].lay_number := -1;
   List[4].Entry_Points[7].operation_type := 'transfer_slot2out';
   List[4].Entry_Points[7].part_destination := '';
   List[4].Entry_Points[7].part_status := 'gripper';
   List[4].Entry_Points[7].robot_status := 'home';
   List[4].Entry_Points[7].machine_status := '';
   List[4].Entry_Points[7].previous_trajectory := 'TakeFromSlot';
   List[4].Entry_Points[7].active := true;
   List[3].Entry_Points[3].part_side := '';
   List[3].Entry_Points[3].operation_side := '';
   List[3].Entry_Points[3].lay_number := -1;
   List[3].Entry_Points[3].operation_type := 'transfer_in2slot';
   List[3].Entry_Points[3].part_destination := 'part_slot';
   List[3].Entry_Points[3].part_status := 'gripper';
   List[3].Entry_Points[3].robot_status := 'pallet_in';
   List[3].Entry_Points[3].machine_status := '';
   List[3].Entry_Points[3].previous_trajectory := 'TakeFromPalletIn';
   List[3].Entry_Points[3].active := true;
   List[2].Entry_Points[1].operation_type := 'machining';
   List[2].Entry_Points[1].lay_number := -1;
   List[2].Entry_Points[1].operation_side := 'B';
   List[2].Entry_Points[1].part_side := 'B';
   List[2].Entry_Points[2].active := true;
   List[2].Entry_Points[2].previous_trajectory := 'AutoMachiningA_';
   List[2].Entry_Points[2].machine_status := 'ready2load';
   List[2].Entry_Points[2].robot_status := 'flip_table';
   List[2].Entry_Points[2].part_status := 'flip_table';
   List[2].Entry_Points[2].part_destination := 'pallet_out';
   List[2].Entry_Points[2].operation_type := 'machining';
   List[2].Entry_Points[2].lay_number := -1;
   List[2].Entry_Points[2].operation_side := 'B';
   List[2].Entry_Points[2].part_side := 'B';
   List[15].Entry_Points[1].active := true;
   List[15].Entry_Points[1].previous_trajectory := 'Pallet_Scanning';
   List[15].Entry_Points[1].machine_status := 'ready2load';
   List[15].Entry_Points[1].robot_status := 'home';
   List[15].Entry_Points[1].part_status := 'pallet_in';
   List[15].Entry_Points[1].part_destination := 'pallet_out';
   List[6].Entry_Points[9].part_side := 'A';
   List[6].Entry_Points[9].operation_side := 'A';
   List[6].Entry_Points[9].lay_number := -1;
   List[6].Entry_Points[9].operation_type := 'machining';
   List[6].Entry_Points[9].part_destination := '';
   List[6].Entry_Points[9].part_status := 'flip_table';
   List[6].Entry_Points[9].robot_status := 'flip_table';
   List[6].Entry_Points[9].machine_status := 'ready2load';
   List[6].Entry_Points[9].previous_trajectory := 'PutOnFlipTableB';
   List[6].Entry_Points[9].active := true;
   List[5].Entry_Points[4].part_side := 'B';
   List[5].Entry_Points[4].operation_side := 'B';
   List[5].Entry_Points[4].lay_number := -1;
   List[5].Entry_Points[4].operation_type := 'transfer_in2out';
   List[5].Entry_Points[4].part_destination := '';
   List[5].Entry_Points[4].part_status := 'gripper';
   List[5].Entry_Points[4].robot_status := 'pallet_in';
   List[5].Entry_Points[4].machine_status := '';
   List[5].Entry_Points[4].previous_trajectory := 'TakeFromPalletIn';
   List[5].Entry_Points[4].active := true;
   List[5].Entry_Points[3].part_side := 'B';
   List[5].Entry_Points[3].operation_side := 'B';
   List[5].Entry_Points[3].lay_number := -1;
   List[5].Entry_Points[3].operation_type := 'machining';
   List[5].Entry_Points[3].part_destination := '';
   List[5].Entry_Points[3].part_status := 'gripper';
   List[5].Entry_Points[3].robot_status := 'pallet_in';
   List[5].Entry_Points[3].machine_status := '';
   List[5].Entry_Points[3].previous_trajectory := 'TakeFromPalletIn';
   List[5].Entry_Points[3].active := true;
   List[4].Entry_Points[6].part_side := '';
   List[4].Entry_Points[6].operation_side := '';
   List[4].Entry_Points[6].lay_number := -1;
   List[4].Entry_Points[6].operation_type := 'transfer_in2out';
   List[4].Entry_Points[6].part_destination := '';
   List[4].Entry_Points[6].part_status := 'gripper';
   List[4].Entry_Points[6].robot_status := 'pallet_in';
   List[4].Entry_Points[6].machine_status := '';
   List[4].Entry_Points[6].previous_trajectory := 'AutoMachiningA_';
   List[4].Entry_Points[6].active := true;
   List[6].Entry_Points[8].part_side := '';
   List[6].Entry_Points[8].operation_side := '';
   List[6].Entry_Points[8].lay_number := -1;
   List[6].Entry_Points[8].operation_type := 'machining';
   List[6].Entry_Points[8].part_destination := '';
   List[6].Entry_Points[8].part_status := 'flip_table';
   List[6].Entry_Points[8].robot_status := 'home';
   List[6].Entry_Points[8].machine_status := '';
   List[6].Entry_Points[8].previous_trajectory := 'PutOnFlipTableA';
   List[6].Entry_Points[8].active := true;
   List[1].Entry_Points[4].part_side := '';
   List[1].Entry_Points[4].operation_side := '';
   List[1].Entry_Points[4].lay_number := -1;
   List[1].Entry_Points[4].operation_type := 'scanning';
   List[1].Entry_Points[4].part_destination := '';
   List[1].Entry_Points[4].part_status := '';
   List[1].Entry_Points[4].robot_status := 'flip_table';
   List[1].Entry_Points[4].machine_status := '';
   List[1].Entry_Points[4].previous_trajectory := '';
   List[1].Entry_Points[4].active := true;
   List[6].Entry_Points[7].active := true;
   List[6].Entry_Points[7].previous_trajectory := 'PutOnFlipTableB';
   List[6].Entry_Points[7].machine_status := 'ready2load';
   List[6].Entry_Points[7].robot_status := 'home';
   List[6].Entry_Points[7].part_status := 'flip_table';
   List[6].Entry_Points[7].part_destination := '';
   List[6].Entry_Points[7].operation_type := 'machining';
   List[6].Entry_Points[7].lay_number := -1;
   List[6].Entry_Points[7].operation_side := 'B';
   List[6].Entry_Points[7].part_side := 'B';
   List[10].Entry_Points[2].part_side := 'A';
   List[10].Entry_Points[2].operation_side := 'B';
   List[10].Entry_Points[2].lay_number := -1;
   List[10].Entry_Points[2].operation_type := 'machining';
   List[10].Entry_Points[2].part_destination := 'pallet_out';
   List[10].Entry_Points[2].part_status := 'gripper';
   List[10].Entry_Points[2].robot_status := 'pallet_in';
   List[10].Entry_Points[2].machine_status := '';
   List[10].Entry_Points[2].previous_trajectory := 'TakeFromPalletIn';
   List[10].Entry_Points[2].active := true;
   List[6].Entry_Points[6].part_side := 'B';
   List[6].Entry_Points[6].operation_side := 'B';
   List[6].Entry_Points[6].lay_number := -1;
   List[6].Entry_Points[6].operation_type := 'machining';
   List[13].trajectory := 'PutOnFlipTableB';
   List[13].Entry_Points[1].part_side := '';
   List[13].Entry_Points[1].operation_side := '';
   List[13].Entry_Points[1].lay_number := -1;
   List[13].Entry_Points[1].operation_type := 'machining';
   List[13].Entry_Points[1].part_destination := 'flip_table';
   List[13].Entry_Points[1].part_status := 'gripper';
   List[13].Entry_Points[1].robot_status := 'pallet_out';
   List[13].Entry_Points[1].machine_status := '';
   List[13].Entry_Points[1].previous_trajectory := 'UnloadMachine';
   List[13].Entry_Points[1].active := true;
   List[11].Entry_Points[1].part_side := '';
   List[11].Entry_Points[1].operation_side := '';
   List[11].Entry_Points[1].lay_number := -1;
   List[11].Entry_Points[1].operation_type := 'transfer_in2flip';
   List[11].Entry_Points[1].part_destination := '';
   List[11].Entry_Points[1].part_status := 'gripper';
   List[11].Entry_Points[1].robot_status := 'pallet_in';
   List[11].Entry_Points[1].machine_status := '';
   List[11].Entry_Points[1].previous_trajectory := 'TakeFromPalletIn';
   List[11].Entry_Points[1].active := true;
   List[7].Entry_Points[2].part_destination := '';
   List[6].Entry_Points[5].part_status := 'flip_table';
   List[6].Entry_Points[4].part_destination := '';
   List[5].Entry_Points[2].part_side := 'A';
   List[5].Entry_Points[2].operation_side := 'A';
   List[5].Entry_Points[2].lay_number := -1;
   List[5].Entry_Points[2].operation_type := 'machining';
   List[12].OUT_Status.inprocess_part_status := 'pallet_in';
   List[12].OUT_Status.finish_part_status := 'pallet_in';
   List[15].Entry_Points[1].operation_type := 'machining';
   List[15].Entry_Points[1].lay_number := -1;
   List[15].Entry_Points[1].operation_side := 'A';
   List[15].Entry_Points[1].part_side := 'A';
   List[15].Entry_Points[3].active := true;
   List[15].Entry_Points[3].previous_trajectory := 'PartHeightMeasuring';
   List[15].Entry_Points[3].machine_status := 'ready2load';
   List[15].Entry_Points[3].robot_status := 'pallet_in';
   List[15].Entry_Points[3].part_status := 'pallet_in';
   List[15].Entry_Points[3].part_destination := 'pallet_out';
   List[9].Entry_Points[5].part_destination := '';
   List[9].Entry_Points[4].part_destination := '';
   List[15].Entry_Points[3].operation_type := 'machining';
   List[15].Entry_Points[3].lay_number := -1;
   List[15].Entry_Points[3].operation_side := 'A';
   List[15].Entry_Points[3].part_side := 'A';
   List[15].Entry_Points[2].active := true;
   List[15].Entry_Points[2].previous_trajectory := 'AutoMachiningA';
   List[15].Entry_Points[2].machine_status := 'ready2load';
   List[15].Entry_Points[2].robot_status := 'pallet_out';
   List[15].Entry_Points[2].part_status := 'pallet_in';
   List[15].Entry_Points[2].part_destination := 'pallet_out';
   List[15].Entry_Points[2].operation_type := 'machining';
   List[15].Entry_Points[2].lay_number := -1;
   List[15].Entry_Points[2].operation_side := 'A';
   List[15].Entry_Points[2].part_side := 'A';
   List[1].Entry_Points[3].part_side := '';
   List[1].Entry_Points[3].operation_side := '';
   List[1].Entry_Points[3].lay_number := -1;
   List[1].Entry_Points[3].operation_type := 'scanning';
   List[1].Entry_Points[3].part_destination := '';
   List[1].Entry_Points[3].part_status := '';
   List[1].Entry_Points[3].robot_status := 'pallet_out';
   List[1].Entry_Points[3].machine_status := '';
   List[1].Entry_Points[3].previous_trajectory := '';
   List[1].Entry_Points[3].active := true;
   List[12].Entry_Points[1].part_side := '';
   List[12].Entry_Points[1].operation_side := '';
   List[12].Entry_Points[1].lay_number := -1;
   List[12].Entry_Points[1].operation_type := 'go_home';
   List[12].Entry_Points[1].part_destination := '';
   List[12].Entry_Points[1].part_status := '';
   List[12].Entry_Points[1].machine_status := '';
   List[12].Entry_Points[1].previous_trajectory := '';
   List[12].Entry_Points[1].active := true;
   List[12].OUT_Status.finish_task_status := 'done';
   List[12].OUT_Status.inprocess_task_status := 'in_process';
   List[12].trajectory := 'go_home';
   List[9].Entry_Points[3].part_destination := '';
   List[1].Entry_Points[2].part_side := '';
   List[1].Entry_Points[2].operation_side := '';
   List[1].Entry_Points[2].lay_number := -1;
   List[1].Entry_Points[2].operation_type := 'scanning';
   List[1].Entry_Points[2].part_destination := '';
   List[1].Entry_Points[2].part_status := '';
   List[1].Entry_Points[2].robot_status := 'pallet_in';
   List[1].Entry_Points[2].machine_status := '';
   List[1].Entry_Points[2].previous_trajectory := '';
   List[1].Entry_Points[2].active := true;
   List[11].OUT_Status.finish_part_status := 'flip_table';
   List[11].OUT_Status.finish_task_status := 'done';
   List[11].OUT_Status.inprocess_part_status := 'dropping';
   List[11].OUT_Status.inprocess_task_status := 'in_process';
   List[10].Entry_Points[7].operation_side := '';
   List[10].Entry_Points[7].part_side := '';
   List[11].trajectory := 'PutOnFlipTableA';
   List[6].Entry_Points[2].part_destination := '';
   List[4].Entry_Points[2].part_destination := 'pallet_out';
   List[5].Entry_Points[1].part_destination := '';
   List[5].Entry_Points[2].active := true;
   List[11].Entry_Points[5].part_side := '';
   List[11].Entry_Points[5].operation_side := '';
   List[11].Entry_Points[5].lay_number := -1;
   List[11].Entry_Points[5].operation_type := '';
   List[11].Entry_Points[5].part_destination := '';
   List[11].Entry_Points[5].part_status := '';
   List[11].Entry_Points[5].robot_status := '';
   List[11].Entry_Points[5].machine_status := '';
   List[11].Entry_Points[5].previous_trajectory := '';
   List[11].Entry_Points[5].active := false;
   List[11].Entry_Points[4].part_side := '';
   List[11].Entry_Points[4].operation_side := '';
   List[11].Entry_Points[4].lay_number := -1;
   List[11].Entry_Points[4].operation_type := '';
   List[11].Entry_Points[4].part_destination := '';
   List[11].Entry_Points[4].part_status := '';
   List[11].Entry_Points[4].robot_status := '';
   List[11].Entry_Points[4].machine_status := '';
   List[11].Entry_Points[4].previous_trajectory := '';
   List[11].Entry_Points[4].active := false;
   List[11].Entry_Points[3].part_side := '';
   List[11].Entry_Points[3].operation_side := '';
   List[11].Entry_Points[3].lay_number := -1;
   List[11].Entry_Points[3].operation_type := '';
   List[11].Entry_Points[3].part_destination := '';
   List[11].Entry_Points[3].part_status := '';
   List[11].Entry_Points[3].robot_status := '';
   List[11].Entry_Points[3].machine_status := '';
   List[11].Entry_Points[3].previous_trajectory := '';
   List[11].Entry_Points[3].active := false;
   List[11].Entry_Points[2].part_side := ' ';
   List[11].Entry_Points[2].operation_side := ' ';
   List[11].Entry_Points[2].lay_number := -1;
   List[11].Entry_Points[2].operation_type := '';
   List[11].Entry_Points[2].part_destination := '';
   List[11].Entry_Points[2].part_status := '';
   List[11].Entry_Points[2].robot_status := '';
   List[11].Entry_Points[2].machine_status := '';
   List[11].Entry_Points[2].previous_trajectory := '';
   List[11].Entry_Points[2].active := false;
   List[10].OUT_Status.finish_part_status := 'flip_table';
   List[10].OUT_Status.finish_task_status := 'on_trajectory';
   List[10].OUT_Status.inprocess_part_status := 'dropping';
   List[10].OUT_Status.inprocess_task_status := 'in_process';
   List[10].Entry_Points[5].part_destination := '';
   List[10].Entry_Points[4].part_destination := 'pallet_out';
   List[10].Entry_Points[3].part_side := 'B';
   List[10].Entry_Points[3].operation_side := 'A';
   List[10].Entry_Points[3].lay_number := -1;
   List[10].Entry_Points[3].operation_type := 'machining';
   List[10].Entry_Points[3].part_destination := 'part_slot';
   List[10].Entry_Points[3].part_status := 'gripper';
   List[10].Entry_Points[3].robot_status := 'pallet_in';
   List[10].Entry_Points[3].machine_status := '';
   List[10].Entry_Points[3].previous_trajectory := 'TakeFromPalletIn';
   List[10].Entry_Points[3].active := true;
   List[13].OUT_Status.inprocess_task_status := 'in_process';
   List[13].OUT_Status.inprocess_part_status := 'dropping';
   List[13].OUT_Status.finish_task_status := 'done';
   List[13].OUT_Status.finish_part_status := 'flip_table';
   List[6].Entry_Points[6].active := true;
   List[6].Entry_Points[6].previous_trajectory := '';
   List[6].Entry_Points[6].machine_status := 'ready2load';
   List[6].Entry_Points[6].robot_status := 'flip_table';
   List[6].Entry_Points[6].part_status := 'flip_table';
   List[6].Entry_Points[6].part_destination := '';
   List[10].Entry_Points[1].part_side := 'A';
   List[10].Entry_Points[1].operation_side := 'B';
   List[10].Entry_Points[1].lay_number := -1;
   List[10].Entry_Points[1].operation_type := 'machining';
   List[10].Entry_Points[1].part_destination := 'part_slot';
   List[10].Entry_Points[1].part_status := 'gripper';
   List[10].Entry_Points[1].robot_status := 'pallet_in';
   List[10].Entry_Points[1].machine_status := '';
   List[10].Entry_Points[1].previous_trajectory := 'TakeFromPalletIn';
   List[10].Entry_Points[1].active := true;
   List[10].trajectory := 'PutOnFlipTableB';
   List[3].Entry_Points[2].part_destination := 'part_slot';
   List[3].Entry_Points[1].part_destination := 'part_slot';
   List[10].Entry_Points[5].part_side := '';
   List[10].Entry_Points[5].operation_side := '';
   List[10].Entry_Points[5].lay_number := -1;
   List[10].Entry_Points[5].operation_type := '';
   List[10].Entry_Points[5].part_status := '';
   List[10].Entry_Points[5].robot_status := '';
   List[10].Entry_Points[5].machine_status := '';
   List[10].Entry_Points[5].previous_trajectory := '';
   List[10].Entry_Points[5].active := false;
   List[10].Entry_Points[4].part_side := 'B';
   List[10].Entry_Points[4].operation_side := 'A';
   List[10].Entry_Points[4].lay_number := -1;
   List[10].Entry_Points[4].operation_type := 'machining';
   List[10].Entry_Points[4].part_status := 'gripper';
   List[10].Entry_Points[4].robot_status := 'pallet_in';
   List[10].Entry_Points[4].machine_status := '';
   List[10].Entry_Points[4].previous_trajectory := 'TakeFromPalletIn';
   List[10].Entry_Points[4].active := true;
   List[3].Entry_Points[5].part_side := '';
   List[3].Entry_Points[5].operation_side := '';
   List[3].Entry_Points[5].lay_number := -1;
   List[3].Entry_Points[5].operation_type := '';
   List[3].Entry_Points[5].part_status := '';
   List[3].Entry_Points[5].robot_status := '';
   List[3].Entry_Points[5].machine_status := '';
   List[3].Entry_Points[5].previous_trajectory := '';
   List[3].Entry_Points[5].active := false;
   List[3].Entry_Points[4].part_side := '';
   List[3].Entry_Points[4].operation_side := '';
   List[3].Entry_Points[4].lay_number := -1;
   List[3].Entry_Points[4].operation_type := '';
   List[3].Entry_Points[4].part_status := '';
   List[3].Entry_Points[4].robot_status := '';
   List[3].Entry_Points[4].machine_status := '';
   List[3].Entry_Points[4].previous_trajectory := '';
   List[3].Entry_Points[4].active := false;
   List[9].Entry_Points[5].part_side := '';
   List[9].Entry_Points[5].operation_side := '';
   List[9].Entry_Points[5].lay_number := -1;
   List[9].Entry_Points[5].operation_type := 'machining';
   List[9].Entry_Points[5].part_status := 'part_slot';
   List[9].Entry_Points[5].robot_status := 'pallet_out';
   List[9].Entry_Points[5].machine_status := '';
   List[9].Entry_Points[5].previous_trajectory := '';
   List[9].Entry_Points[5].active := true;
   List[9].Entry_Points[4].part_side := '';
   List[9].Entry_Points[4].operation_side := '';
   List[9].Entry_Points[4].lay_number := -1;
   List[9].Entry_Points[4].operation_type := 'transfer_slot2out';
   List[9].Entry_Points[4].part_status := 'part_slot';
   List[9].Entry_Points[4].robot_status := 'pallet_out';
   List[9].Entry_Points[4].machine_status := '';
   List[9].Entry_Points[4].previous_trajectory := '';
   List[9].Entry_Points[4].active := true;
   List[9].Entry_Points[3].part_side := '';
   List[9].Entry_Points[3].operation_side := '';
   List[9].Entry_Points[3].lay_number := -1;
   List[9].Entry_Points[3].operation_type := 'transfer_slot2out';
   List[9].Entry_Points[3].part_status := 'part_slot';
   List[9].Entry_Points[3].robot_status := 'pallet_in';
   List[9].Entry_Points[3].machine_status := '';
   List[9].Entry_Points[3].previous_trajectory := '';
   List[9].Entry_Points[3].active := true;
   List[9].Entry_Points[2].part_side := '';
   List[9].Entry_Points[2].operation_side := '';
   List[9].Entry_Points[2].lay_number := -1;
   List[9].Entry_Points[2].operation_type := 'machining';
   List[9].Entry_Points[2].part_status := 'part_slot';
   List[9].Entry_Points[2].robot_status := 'home';
   List[9].Entry_Points[2].machine_status := '';
   List[9].Entry_Points[2].previous_trajectory := '';
   List[9].Entry_Points[2].active := true;
   List[9].Entry_Points[1].part_side := '';
   List[9].Entry_Points[1].operation_side := '';
   List[9].Entry_Points[1].lay_number := -1;
   List[9].Entry_Points[1].operation_type := 'transfer_slot2out';
   List[9].Entry_Points[1].part_status := 'part_slot';
   List[9].Entry_Points[1].robot_status := 'home';
   List[9].Entry_Points[1].machine_status := '';
   List[9].Entry_Points[1].previous_trajectory := '';
   List[9].Entry_Points[1].active := true;
   List[8].Entry_Points[5].part_side := '';
   List[8].Entry_Points[5].operation_side := '';
   List[8].Entry_Points[5].lay_number := -1;
   List[8].Entry_Points[5].operation_type := '';
   List[8].Entry_Points[5].part_status := '';
   List[8].Entry_Points[5].robot_status := '';
   List[8].Entry_Points[5].machine_status := '';
   List[8].Entry_Points[5].previous_trajectory := '';
   List[8].Entry_Points[5].active := false;
   List[8].Entry_Points[4].part_side := '';
   List[8].Entry_Points[4].operation_side := '';
   List[8].Entry_Points[4].lay_number := -1;
   List[8].Entry_Points[4].operation_type := '';
   List[8].Entry_Points[4].part_status := '';
   List[8].Entry_Points[4].robot_status := '';
   List[8].Entry_Points[4].machine_status := '';
   List[8].Entry_Points[4].previous_trajectory := '';
   List[8].Entry_Points[4].active := false;
   List[8].Entry_Points[3].part_side := '';
   List[8].Entry_Points[3].operation_side := '';
   List[8].Entry_Points[3].lay_number := -1;
   List[8].Entry_Points[3].operation_type := '';
   List[8].Entry_Points[3].part_status := '';
   List[8].Entry_Points[3].robot_status := '';
   List[8].Entry_Points[3].machine_status := '';
   List[8].Entry_Points[3].previous_trajectory := '';
   List[8].Entry_Points[3].active := false;
   List[8].Entry_Points[2].part_side := '';
   List[8].Entry_Points[2].operation_side := '';
   List[8].Entry_Points[2].machine_status := '';
   List[8].Entry_Points[1].part_side := '';
   List[8].Entry_Points[1].operation_side := '';
   List[8].Entry_Points[1].machine_status := 'ready2unload';
   List[1].Entry_Points[1].operation_type := 'scanning';
   List[7].Entry_Points[5].part_side := '';
   List[7].Entry_Points[5].operation_side := '';
   List[7].Entry_Points[5].lay_number := -1;
   List[7].Entry_Points[5].operation_type := '';
   List[7].Entry_Points[5].part_status := '';
   List[7].Entry_Points[5].robot_status := '';
   List[7].Entry_Points[5].machine_status := '';
   List[7].Entry_Points[5].previous_trajectory := '';
   List[7].Entry_Points[5].active := false;
   List[7].Entry_Points[3].part_side := '';
   List[7].Entry_Points[3].operation_side := '';
   List[7].Entry_Points[3].lay_number := -1;
   List[7].Entry_Points[3].operation_type := 'machining';
   List[7].Entry_Points[3].part_status := 'gripper';
   List[7].Entry_Points[3].robot_status := 'flip_table';
   List[7].Entry_Points[3].machine_status := 'ready2load';
   List[7].Entry_Points[3].previous_trajectory := 'TakeFromSlot';
   List[7].Entry_Points[3].active := true;
   List[7].Entry_Points[2].part_side := 'B';
   List[7].Entry_Points[2].operation_side := 'B';
   List[7].Entry_Points[2].lay_number := -1;
   List[7].Entry_Points[2].operation_type := 'machining';
   List[7].Entry_Points[2].part_status := 'gripper';
   List[7].Entry_Points[2].robot_status := 'flip_table';
   List[7].Entry_Points[2].machine_status := 'ready2load';
   List[7].Entry_Points[2].previous_trajectory := 'TakeFromFlipTableA';
   List[7].Entry_Points[2].active := true;
   List[7].Entry_Points[1].part_side := 'A';
   List[7].Entry_Points[1].operation_side := 'A';
   List[7].Entry_Points[1].lay_number := -1;
   List[0].OUT_Status.finish_task_status := 'unknown';
   List[0].OUT_Status.finish_part_status := 'unknown';
   List[6].Entry_Points[5].active := true;
   List[6].Entry_Points[5].previous_trajectory := 'PutOnFlipTableA';
   List[6].Entry_Points[5].machine_status := 'ready2load';
   List[6].Entry_Points[5].robot_status := 'flip_table';
   List[6].Entry_Points[5].part_destination := '';
   List[6].Entry_Points[5].operation_type := 'machining';
   List[6].Entry_Points[5].lay_number := -1;
   List[6].Entry_Points[5].operation_side := 'B';
   List[6].Entry_Points[5].part_side := 'B';
   List[6].Entry_Points[4].part_side := '';
   List[6].Entry_Points[4].operation_side := '';
   List[6].Entry_Points[4].lay_number := -1;
   List[6].Entry_Points[4].operation_type := 'transfer_in2out';
   List[6].Entry_Points[4].part_status := 'flip_table';
   List[6].Entry_Points[4].robot_status := 'flip_table';
   List[6].Entry_Points[4].machine_status := '';
   List[6].Entry_Points[4].previous_trajectory := 'PutOnFlipTableA';
   List[6].Entry_Points[4].active := true;
   List[6].Entry_Points[3].part_side := '';
   List[6].Entry_Points[3].operation_side := '';
   List[6].Entry_Points[3].lay_number := -1;
   List[6].Entry_Points[3].operation_type := 'machining';
   List[6].Entry_Points[3].part_status := 'flip_table';
   List[6].Entry_Points[3].robot_status := 'flip_table';
   List[6].Entry_Points[3].machine_status := '';
   List[6].Entry_Points[3].previous_trajectory := 'PutOnFlipTableB';
   List[6].Entry_Points[3].active := true;
   List[6].Entry_Points[2].part_side := '';
   List[6].Entry_Points[2].operation_side := '';
   List[6].Entry_Points[2].lay_number := -1;
   List[6].Entry_Points[1].part_side := 'A';
   List[6].Entry_Points[1].operation_side := 'A';
   List[6].Entry_Points[1].lay_number := -1;
   List[5].Entry_Points[5].part_side := '';
   List[5].Entry_Points[5].operation_side := '';
   List[5].Entry_Points[5].lay_number := -1;
   List[5].Entry_Points[5].operation_type := '';
   List[5].Entry_Points[5].part_status := '';
   List[5].Entry_Points[5].robot_status := '';
   List[5].Entry_Points[5].machine_status := '';
   List[5].Entry_Points[5].previous_trajectory := '';
   List[5].Entry_Points[5].active := false;
   List[6].Entry_Points[3].part_destination := '';
   List[4].Entry_Points[4].part_destination := '';
   List[4].Entry_Points[5].part_destination := '';
   List[5].Entry_Points[2].previous_trajectory := 'TakeFromPalletIn';
   List[5].Entry_Points[2].machine_status := '';
   List[5].Entry_Points[2].robot_status := 'pallet_in';
   List[5].Entry_Points[2].part_status := 'gripper';
   List[5].Entry_Points[2].part_destination := '';
   List[5].Entry_Points[1].lay_number := -1;
   List[4].Entry_Points[5].part_side := '';
   List[4].Entry_Points[5].operation_side := '';
   List[4].Entry_Points[5].lay_number := -1;
   List[4].Entry_Points[5].operation_type := 'transfer_slot2out';
   List[4].Entry_Points[5].part_status := 'gripper';
   List[4].Entry_Points[5].robot_status := 'part_slot';
   List[4].Entry_Points[5].machine_status := '';
   List[4].Entry_Points[5].previous_trajectory := 'TakeFromSlot';
   List[4].Entry_Points[5].active := true;
   List[4].Entry_Points[4].part_side := '';
   List[4].Entry_Points[4].operation_side := '';
   List[4].Entry_Points[4].lay_number := -1;
   List[4].Entry_Points[4].operation_type := 'machining';
   List[4].Entry_Points[4].part_status := 'gripper';
   List[4].Entry_Points[4].robot_status := 'pallet_in';
   List[4].Entry_Points[4].machine_status := '';
   List[4].Entry_Points[4].previous_trajectory := 'PutOnPalletOut';
   List[4].Entry_Points[4].active := true;
   List[4].Entry_Points[3].part_side := '';
   List[4].Entry_Points[3].operation_side := '';
   List[4].Entry_Points[3].lay_number := -1;
   List[4].Entry_Points[3].operation_type := 'transfer_slot2out';
   List[4].Entry_Points[3].part_status := 'gripper';
   List[4].Entry_Points[3].robot_status := 'flip_table';
   List[4].Entry_Points[3].machine_status := '';
   List[4].Entry_Points[3].previous_trajectory := 'TakeFromSlot';
   List[4].Entry_Points[3].active := true;
   List[4].Entry_Points[2].part_side := '';
   List[4].Entry_Points[2].operation_side := '';
   List[4].Entry_Points[2].lay_number := -1;
   List[4].Entry_Points[2].operation_type := 'machining';
   List[4].Entry_Points[2].part_status := 'gripper';
   List[4].Entry_Points[2].robot_status := 'pallet_out';
   List[4].Entry_Points[2].machine_status := '';
   List[4].Entry_Points[2].previous_trajectory := 'UnloadMachine';
   List[4].Entry_Points[2].active := true;
   List[4].Entry_Points[1].lay_number := -1;
   List[8].Entry_Points[2].part_status := '';
   List[8].Entry_Points[2].robot_status := '';
   List[8].Entry_Points[1].part_status := 'in_machine';
   List[8].Entry_Points[1].previous_trajectory := 'LoadMachine';
   List[8].Entry_Points[1].operation_type := 'machining';
   List[8].Entry_Points[1].lay_number := -1;
   List[8].Entry_Points[1].active := true;
   List[8].Entry_Points[2].lay_number := -1;
   List[8].Entry_Points[2].operation_type := '';
   List[8].Entry_Points[2].active := false;
   List[7].Entry_Points[1].part_status := 'gripper';
   List[7].Entry_Points[1].robot_status := 'flip_table';
   List[7].Entry_Points[1].machine_status := 'ready2load';
   List[7].Entry_Points[1].previous_trajectory := 'TakeFromFlipTableA';
   List[7].Entry_Points[1].active := true;
   List[7].Entry_Points[1].operation_type := 'machining';
   List[6].Entry_Points[1].operation_type := 'machining';
   List[6].Entry_Points[2].operation_type := 'machining';
   List[6].Entry_Points[2].previous_trajectory := 'PutOnFlipTableA';
   List[6].Entry_Points[1].previous_trajectory := 'PutOnFlipTableA';
   List[6].Entry_Points[2].part_status := 'flip_table';
   List[6].Entry_Points[2].robot_status := 'flip_table';
   List[6].Entry_Points[2].machine_status := '';
   List[6].Entry_Points[1].part_status := 'flip_table';
   List[6].Entry_Points[1].robot_status := 'flip_table';
   List[6].Entry_Points[1].machine_status := 'ready2load';
   List[6].Entry_Points[2].active := true;
   List[6].Entry_Points[1].active := true;
   List[4].Entry_Points[1].operation_type := 'transfer_in2out';
   List[5].Entry_Points[1].operation_type := 'transfer_in2out';
   List[5].Entry_Points[1].part_status := 'gripper';
   List[5].Entry_Points[1].robot_status := 'pallet_in';
   List[5].Entry_Points[1].machine_status := '';
   List[5].Entry_Points[1].part_side := 'A';
   List[5].Entry_Points[1].operation_side := 'A';
   List[5].Entry_Points[1].previous_trajectory := 'TakeFromPalletIn';
   List[6].OUT_Status.finish_part_status := 'gripper';
   List[6].OUT_Status.finish_task_status := 'on_trajectory';
   List[6].OUT_Status.inprocess_part_status := 'flipping';
   List[6].OUT_Status.inprocess_task_status := 'in_process';
   List[8].Entry_Points[2].previous_trajectory := '';
   List[5].OUT_Status.finish_part_status := 'flip_table';
   List[5].OUT_Status.finish_task_status := 'on_trajectory';
   List[5].OUT_Status.inprocess_part_status := 'dropping';
   List[5].OUT_Status.inprocess_task_status := 'in_process';
   List[4].OUT_Status.finish_part_status := 'pallet_out';
   List[4].OUT_Status.finish_task_status := 'done';
   List[4].OUT_Status.inprocess_part_status := 'dropping';
   List[4].OUT_Status.inprocess_task_status := 'in_process';
   List[4].trajectory := 'PutOnPalletOut';
   List[3].Entry_Points[1].lay_number := -1;
   List[8].Entry_Points[1].robot_status := 'at_machine';
   List[3].Entry_Points[1].machine_status := '';
   List[3].Entry_Points[1].operation_side := '';
   List[3].Entry_Points[1].part_side := '';
   List[3].Entry_Points[2].lay_number := -1;
   List[3].Entry_Points[2].machine_status := '';
   List[3].Entry_Points[2].previous_trajectory := 'UnloadMachine';
   List[3].Entry_Points[2].active := true;
   List[9].trajectory := 'TakeFromSlot';
   List[3].Entry_Points[1].active := true;
   List[3].Entry_Points[2].part_side := '';
   List[3].Entry_Points[1].robot_status := 'flip_table';
   List[4].Entry_Points[1].machine_status := '';
   List[4].Entry_Points[1].robot_status := 'pallet_in';
   List[4].Entry_Points[1].part_status := 'gripper';
   List[4].Entry_Points[1].previous_trajectory := 'TakeFromPalletIn';
   List[4].Entry_Points[1].active := true;
   List[4].Entry_Points[1].operation_side := '';
   List[4].Entry_Points[1].part_side := '';
   List[5].Entry_Points[1].active := true;
   List[5].trajectory := 'PutOnFlipTableA';
   List[3].Entry_Points[2].part_status := 'gripper';
   List[9].OUT_Status.inprocess_part_status := 'grabbing';
   List[9].OUT_Status.finish_part_status := 'gripper';
   List[3].Entry_Points[1].operation_type := 'transfer_in2out';
   List[8].OUT_Status.finish_task_status := 'on_trajectory';
   List[8].OUT_Status.inprocess_task_status := 'in_process';
   List[7].OUT_Status.finish_task_status := 'on_trajectory';
   List[7].OUT_Status.inprocess_task_status := 'in_process';
   List[3].OUT_Status.finish_task_status := 'done';
   List[3].OUT_Status.inprocess_task_status := 'in_process';
   List[1].OUT_Status.finish_task_status := 'done';
   List[1].OUT_Status.inprocess_task_status := 'in_process';
   List[9].OUT_Status.finish_task_status := 'on_trajectory';
   List[3].Entry_Points[2].robot_status := 'pallet_out';
   List[8].OUT_Status.inprocess_part_status := 'unloading';
   List[7].OUT_Status.inprocess_part_status := 'loading';
   List[1].OUT_Status.inprocess_part_status := 'pallet_in';
   List[1].Entry_Points[1].robot_status := 'home';
   List[9].OUT_Status.inprocess_task_status := 'in_process';
   List[1].Entry_Points[1].active := true;
   List[3].Entry_Points[1].previous_trajectory := 'TakeFromFlipTableA';
   List[3].Entry_Points[2].operation_side := '';
   List[3].Entry_Points[1].part_status := 'gripper';
   List[3].Entry_Points[2].operation_type := 'machining';
   List[8].trajectory := 'UnloadMachine';
   List[3].OUT_Status.inprocess_part_status := 'dropping';
   List[8].OUT_Status.finish_part_status := 'gripper';
   List[7].trajectory := 'LoadMachine';
   List[7].OUT_Status.finish_part_status := 'in_machine';
   List[6].trajectory := 'TakeFromFlipTableA';
   List[3].trajectory := 'PutOnSlot';
   List[3].OUT_Status.finish_part_status := 'part_slot';
   List[2].trajectory := 'AutoMachining_B';
   List[1].trajectory := 'Pallet_Scanning';
   List[1].OUT_Status.finish_part_status := 'pallet_in';
   List[2].Entry_Points[1].part_destination := 'pallet_out';
   List[2].Entry_Points[1].part_status := 'flip_table';
   List[2].Entry_Points[1].robot_status := 'flip_table';
   List[2].Entry_Points[1].machine_status := 'ready2load';
   List[2].Entry_Points[1].previous_trajectory := 'PutOnFlipTableB';
   List[2].Entry_Points[1].active := true;
   List[15].OUT_Status.finish_part_status := 'pallet_out';
   List[15].OUT_Status.inprocess_part_status := '';
   List[15].OUT_Status.inprocess_task_status := 'in_process';
   List[15].OUT_Status.finish_task_status := 'done';
   List[14].trajectory := 'PartHeightMeasuring';
   List[14].Entry_Points[1].operation_type := 'measuring_height';
   List[14].Entry_Points[1].active := true;
   List[14].Entry_Points[2].operation_type := 'measuring_height';
   List[14].Entry_Points[2].active := true;
   List[14].Entry_Points[1].previous_trajectory := '';
   List[14].Entry_Points[2].previous_trajectory := 'PartHeightMeasuring';
   List[14].Entry_Points[1].robot_status := 'home';
   List[14].Entry_Points[2].robot_status := 'pallet_in';
   List[14].Entry_Points[2].part_status := 'scanned';
   List[14].Entry_Points[1].part_status := 'scanned';
   List[14].OUT_Status.inprocess_task_status := 'in_process';
   List[14].OUT_Status.inprocess_part_status := 'scanned';
   List[14].OUT_Status.finish_task_status := 'done';
   List[14].OUT_Status.finish_part_status := '';
   List[14].Entry_Points[3].active := true;
   List[14].Entry_Points[3].previous_trajectory := 'PartHeightMeasuring';
   List[14].Entry_Points[3].machine_status := '';
   List[14].Entry_Points[3].robot_status := 'pallet_in';
   List[14].Entry_Points[3].part_status := 'pallet_in';
   List[14].Entry_Points[3].part_destination := '';
   List[14].Entry_Points[3].operation_type := 'measuring_height';
   List[14].Entry_Points[4].part_status := 'scanned';
   List[14].Entry_Points[4].operation_type := 'measuring_height';
   List[14].Entry_Points[4].active := true;
   List[17].OUT_Status.inprocess_task_status := 'in_process';
   List[17].OUT_Status.inprocess_part_status := '';
   List[17].OUT_Status.finish_task_status := 'done';
   List[17].OUT_Status.finish_part_status := 'flip_table';
   List[17].trajectory := 'AutoMachiningA_';
   List[17].Entry_Points[1].active := true;
   List[17].Entry_Points[1].previous_trajectory := 'Pallet_Scanning';
   List[17].Entry_Points[1].machine_status := 'ready2load';
   List[17].Entry_Points[1].robot_status := 'home';
   List[17].Entry_Points[1].part_status := 'pallet_in';
   List[17].Entry_Points[1].part_destination := 'flip_table';
   List[17].Entry_Points[1].operation_type := 'machining';
   List[17].Entry_Points[1].lay_number := -1;
   List[17].Entry_Points[1].operation_side := 'A';
   List[17].Entry_Points[1].part_side := 'A';
   List[17].Entry_Points[2].active := true;
   List[17].Entry_Points[2].previous_trajectory := 'PutOnPalletOut';
   List[17].Entry_Points[2].machine_status := 'ready2load';
   List[17].Entry_Points[2].robot_status := 'pallet_in';
   List[17].Entry_Points[2].part_status := 'pallet_in';
   List[17].Entry_Points[2].part_destination := 'flip_table';
   List[17].Entry_Points[2].operation_type := 'machining';
   List[17].Entry_Points[2].lay_number := -1;
   List[17].Entry_Points[2].operation_side := 'A';
   List[17].Entry_Points[2].part_side := 'A';
   List[16].Entry_Points[4].active := true;
   List[16].Entry_Points[4].previous_trajectory := '';
   List[16].Entry_Points[4].machine_status := 'ready2load';
   List[16].Entry_Points[4].robot_status := 'pallet_in';
   List[16].Entry_Points[4].part_status := 'pallet_in';
   List[16].Entry_Points[4].part_destination := 'pallet_out';
   List[16].Entry_Points[4].operation_type := 'machining';
   List[16].Entry_Points[4].lay_number := -1;
   List[16].Entry_Points[4].operation_side := 'B';
   List[16].Entry_Points[4].part_side := 'A';
   List[17].Entry_Points[3].active := true;
   List[17].Entry_Points[3].previous_trajectory := 'AutoMachiningB';
   List[17].Entry_Points[3].machine_status := 'ready2load';
   List[17].Entry_Points[3].robot_status := 'pallet_in';
   List[17].Entry_Points[3].part_status := 'pallet_in';
   List[17].Entry_Points[3].part_destination := 'flip_table';
   List[17].Entry_Points[3].operation_type := 'machining';
   List[17].Entry_Points[3].lay_number := -1;
   List[17].Entry_Points[3].operation_side := 'A';
   List[17].Entry_Points[3].part_side := 'A';
   List[17].Entry_Points[4].active := true;
   List[17].Entry_Points[4].previous_trajectory := 'PartHeightMeasuring';
   List[17].Entry_Points[4].machine_status := 'ready2load';
   List[17].Entry_Points[4].robot_status := 'pallet_in';
   List[17].Entry_Points[4].part_status := 'pallet_in';
   List[17].Entry_Points[4].part_destination := 'flip_table';
   List[17].Entry_Points[4].operation_type := 'machining';
   List[17].Entry_Points[4].lay_number := -1;
   List[17].Entry_Points[4].operation_side := 'A';
   List[17].Entry_Points[4].part_side := 'A';
   List[15].Entry_Points[4].active := true;
   List[15].Entry_Points[4].previous_trajectory := 'AutoMachiningB';
   List[15].Entry_Points[4].machine_status := 'ready2load';
   List[15].Entry_Points[4].robot_status := 'pallet_out';
   List[15].Entry_Points[4].part_status := 'pallet_in';
   List[15].Entry_Points[4].part_destination := 'pallet_out';
   List[15].Entry_Points[4].operation_type := 'machining';
   List[15].Entry_Points[4].lay_number := -1;
   List[15].Entry_Points[4].operation_side := 'A';
   List[15].Entry_Points[4].part_side := 'A';
   List[15].Entry_Points[5].active := true;
   List[15].Entry_Points[5].previous_trajectory := 'AutoMachining_B';
   List[15].Entry_Points[5].machine_status := 'ready2load';
   List[15].Entry_Points[5].robot_status := 'pallet_out';
   List[15].Entry_Points[5].part_status := 'pallet_in';
   List[15].Entry_Points[5].part_destination := 'pallet_out';
   List[15].Entry_Points[5].operation_type := 'machining';
   List[15].Entry_Points[5].lay_number := -1;
   List[15].Entry_Points[5].operation_side := 'A';
   List[15].Entry_Points[5].part_side := 'A';
   List[15].trajectory := 'AutoMachiningA';
   List[16].OUT_Status.inprocess_task_status := 'in_process';
   List[16].OUT_Status.inprocess_part_status := '';
   List[16].OUT_Status.finish_task_status := 'done';
   List[16].OUT_Status.finish_part_status := 'pallet_out';
   List[16].trajectory := 'AutoMachiningB';
   List[16].Entry_Points[1].active := true;
   List[16].Entry_Points[1].previous_trajectory := 'AutoMachiningA';
   List[16].Entry_Points[1].machine_status := 'ready2load';
   List[16].Entry_Points[1].robot_status := 'pallet_out';
   List[16].Entry_Points[1].part_status := 'pallet_in';
   List[16].Entry_Points[1].part_destination := 'pallet_out';
   List[16].Entry_Points[1].operation_type := 'machining';
   List[16].Entry_Points[1].lay_number := -1;
   List[16].Entry_Points[1].operation_side := 'B';
   List[16].Entry_Points[1].part_side := 'A';
   List[16].Entry_Points[2].active := true;
   List[16].Entry_Points[2].previous_trajectory := 'AutoMachiningB';
   List[16].Entry_Points[2].machine_status := 'ready2load';
   List[16].Entry_Points[2].robot_status := 'pallet_out';
   List[16].Entry_Points[2].part_status := 'pallet_in';
   List[16].Entry_Points[2].part_destination := 'pallet_out';
   List[16].Entry_Points[2].operation_type := 'machining';
   List[16].Entry_Points[2].lay_number := -1;
   List[16].Entry_Points[2].operation_side := 'B';
   List[16].Entry_Points[2].part_side := 'A';
   List[16].Entry_Points[3].active := true;
   List[16].Entry_Points[3].previous_trajectory := 'AutoMachining_B';
   List[16].Entry_Points[3].machine_status := 'ready2load';
   List[16].Entry_Points[3].robot_status := 'pallet_out';
   List[16].Entry_Points[3].part_status := 'pallet_in';
   List[16].Entry_Points[3].part_destination := 'pallet_out';
   List[16].Entry_Points[3].operation_type := 'machining';
   List[16].Entry_Points[3].lay_number := -1;
   List[16].Entry_Points[3].operation_side := 'B';
   List[16].Entry_Points[3].part_side := 'A';
   List[18].trajectory := 'TakeFromPalletIn';
   List[18].Entry_Points[1].active := true;
   List[18].Entry_Points[1].previous_trajectory := '';
   List[18].Entry_Points[1].machine_status := 'ready2load';
   List[18].Entry_Points[1].robot_status := 'home';
   List[18].Entry_Points[1].part_status := 'pallet_in';
   List[18].Entry_Points[1].part_destination := '';
   List[18].Entry_Points[1].operation_type := 'machining';
   List[18].Entry_Points[1].lay_number := -1;
   List[18].Entry_Points[1].operation_side := '';
   List[18].Entry_Points[1].part_side := '';
   List[18].Entry_Points[2].active := true;
   List[18].Entry_Points[2].previous_trajectory := '';
   List[18].Entry_Points[2].machine_status := '';
   List[18].Entry_Points[2].robot_status := '';
   List[18].Entry_Points[2].part_status := 'pallet_in';
   List[18].Entry_Points[2].part_destination := '';
   List[18].Entry_Points[2].operation_type := 'transfer_in2out';
   List[18].Entry_Points[2].lay_number := -1;
   List[18].Entry_Points[2].operation_side := '';
   List[18].Entry_Points[2].part_side := '';
   List[18].Entry_Points[3].active := true;
   List[18].Entry_Points[3].previous_trajectory := '';
   List[18].Entry_Points[3].machine_status := '';
   List[18].Entry_Points[3].robot_status := 'home';
   List[18].Entry_Points[3].part_status := 'pallet_in';
   List[18].Entry_Points[3].part_destination := '';
   List[18].Entry_Points[3].operation_type := 'transfer_in2flip';
   List[18].Entry_Points[3].lay_number := -1;
   List[18].Entry_Points[3].operation_side := '';
   List[18].Entry_Points[3].part_side := '';
   List[18].Entry_Points[4].active := true;
   List[18].Entry_Points[4].previous_trajectory := '';
   List[18].Entry_Points[4].machine_status := 'ready2load';
   List[18].Entry_Points[4].robot_status := 'pallet_in';
   List[18].Entry_Points[4].part_status := 'pallet_in';
   List[18].Entry_Points[4].part_destination := '';
   List[18].Entry_Points[4].operation_type := 'machining';
   List[18].Entry_Points[4].lay_number := -1;
   List[18].Entry_Points[4].operation_side := '';
   List[18].Entry_Points[4].part_side := '';
   List[18].Entry_Points[5].active := true;
   List[18].Entry_Points[5].previous_trajectory := '';
   List[18].Entry_Points[5].machine_status := '';
   List[18].Entry_Points[5].robot_status := 'pallet_in';
   List[18].Entry_Points[5].part_status := 'pallet_in';
   List[18].Entry_Points[5].part_destination := '';
   List[18].Entry_Points[5].operation_type := 'transfer_in2flip';
   List[18].Entry_Points[5].lay_number := -1;
   List[18].Entry_Points[5].operation_side := '';
   List[18].Entry_Points[5].part_side := '';
   List[18].Entry_Points[6].active := true;
   List[18].Entry_Points[6].previous_trajectory := '';
   List[18].Entry_Points[6].machine_status := 'ready2load';
   List[18].Entry_Points[6].robot_status := 'pallet_out';
   List[18].Entry_Points[6].part_status := 'pallet_in';
   List[18].Entry_Points[6].part_destination := '';
   List[18].Entry_Points[6].operation_type := 'machining';
   List[18].Entry_Points[6].lay_number := -1;
   List[18].Entry_Points[6].operation_side := '';
   List[18].Entry_Points[6].part_side := '';
   List[18].Entry_Points[7].active := true;
   List[18].Entry_Points[7].previous_trajectory := '';
   List[18].Entry_Points[7].machine_status := '';
   List[18].Entry_Points[7].robot_status := 'pallet_out';
   List[18].Entry_Points[7].part_status := '';
   List[18].Entry_Points[7].part_destination := '';
   List[18].Entry_Points[7].operation_type := 'transfer_in2out';
   List[18].Entry_Points[7].lay_number := -1;
   List[18].Entry_Points[7].operation_side := '';
   List[18].Entry_Points[7].part_side := '';
   List[18].Entry_Points[8].active := true;
   List[18].Entry_Points[8].previous_trajectory := '';
   List[18].Entry_Points[8].machine_status := '';
   List[18].Entry_Points[8].robot_status := 'pallet_out';
   List[18].Entry_Points[8].part_status := 'pallet_in';
   List[18].Entry_Points[8].part_destination := '';
   List[18].Entry_Points[8].operation_type := 'transfer_in2flip';
   List[18].Entry_Points[8].lay_number := -1;
   List[18].Entry_Points[8].operation_side := '';
   List[18].Entry_Points[8].part_side := '';
   List[18].Entry_Points[9].active := true;
   List[18].Entry_Points[9].previous_trajectory := '';
   List[18].Entry_Points[9].machine_status := 'ready2load';
   List[18].Entry_Points[9].robot_status := 'flip_table';
   List[18].Entry_Points[9].part_status := 'pallet_in';
   List[18].Entry_Points[9].part_destination := '';
   List[18].Entry_Points[9].operation_type := 'machining';
   List[18].Entry_Points[9].lay_number := -1;
   List[18].Entry_Points[9].operation_side := '';
   List[18].Entry_Points[9].part_side := '';
   List[18].Entry_Points[10].active := true;
   List[18].Entry_Points[10].previous_trajectory := '';
   List[18].Entry_Points[10].machine_status := '';
   List[18].Entry_Points[10].robot_status := 'home';
   List[18].Entry_Points[10].part_status := 'pallet_in';
   List[18].Entry_Points[10].part_destination := '';
   List[18].Entry_Points[10].operation_type := 'transfer_in2slot';
   List[18].Entry_Points[10].lay_number := -1;
   List[18].Entry_Points[10].operation_side := '';
   List[18].Entry_Points[10].part_side := '';
   List[18].Entry_Points[11].active := true;
   List[18].Entry_Points[11].previous_trajectory := '';
   List[18].Entry_Points[11].machine_status := '';
   List[18].Entry_Points[11].robot_status := 'pallet_in';
   List[18].Entry_Points[11].part_status := 'pallet_in';
   List[18].Entry_Points[11].part_destination := '';
   List[18].Entry_Points[11].operation_type := 'transfer_in2slot';
   List[18].Entry_Points[11].lay_number := -1;
   List[18].Entry_Points[11].operation_side := '';
   List[18].Entry_Points[11].part_side := '';
   List[18].Entry_Points[12].active := true;
   List[18].Entry_Points[12].previous_trajectory := '';
   List[18].Entry_Points[12].machine_status := '';
   List[18].Entry_Points[12].robot_status := 'flip_table';
   List[18].Entry_Points[12].part_status := 'pallet_in';
   List[18].Entry_Points[12].part_destination := '';
   List[18].Entry_Points[12].operation_type := 'transfer_in2flip';
   List[18].Entry_Points[12].lay_number := -1;
   List[18].Entry_Points[12].operation_side := '';
   List[18].Entry_Points[12].part_side := '';
   List[18].OUT_Status.inprocess_task_status := 'in_process';
   List[18].OUT_Status.inprocess_part_status := 'grabbing';
   List[18].OUT_Status.finish_task_status := 'on_trajectory';
   List[18].OUT_Status.finish_part_status := 'gripper';
   List[2].OUT_Status.inprocess_task_status := 'in_process';
   List[2].OUT_Status.inprocess_part_status := '';
   List[2].OUT_Status.finish_task_status := 'done';
   List[2].OUT_Status.finish_part_status := 'pallet_out';
   List[15].Entry_Points[6].active := true;
   List[15].Entry_Points[6].previous_trajectory := '';
   List[15].Entry_Points[6].machine_status := 'ready2load';
   List[15].Entry_Points[6].robot_status := 'pallet_in';
   List[15].Entry_Points[6].part_status := 'pallet_in';
   List[15].Entry_Points[6].part_destination := 'pallet_out';
   List[15].Entry_Points[6].operation_type := 'machining';
   List[15].Entry_Points[6].lay_number := -1;
   List[15].Entry_Points[6].operation_side := 'A';
   List[15].Entry_Points[6].part_side := 'A';
   List[16].Entry_Points[5].active := true;
   List[16].Entry_Points[5].previous_trajectory := '';
   List[16].Entry_Points[5].machine_status := 'ready2load';
   List[16].Entry_Points[5].robot_status := 'home';
   List[16].Entry_Points[5].part_status := 'pallet_in';
   List[16].Entry_Points[5].part_destination := 'pallet_out';
   List[16].Entry_Points[5].operation_type := 'machining';
   List[16].Entry_Points[5].lay_number := -1;
   List[16].Entry_Points[5].operation_side := 'B';
   List[16].Entry_Points[5].part_side := 'A';
   List[15].Entry_Points[7].active := true;
   List[15].Entry_Points[7].previous_trajectory := '';
   List[15].Entry_Points[7].machine_status := 'ready2load';
   List[15].Entry_Points[7].robot_status := 'home';
   List[15].Entry_Points[7].part_status := 'pallet_in';
   List[15].Entry_Points[7].part_destination := 'pallet_out';
   List[15].Entry_Points[7].operation_type := 'machining';
   List[15].Entry_Points[7].lay_number := -1;
   List[15].Entry_Points[7].operation_side := 'A';
   List[15].Entry_Points[7].part_side := 'A';
   List[17].Entry_Points[5].active := true;
   List[17].Entry_Points[5].previous_trajectory := 'AutoMachining_B';
   List[17].Entry_Points[5].machine_status := 'ready2load';
   List[17].Entry_Points[5].robot_status := 'pallet_out';
   List[17].Entry_Points[5].part_status := 'pallet_in';
   List[17].Entry_Points[5].part_destination := 'flip_table';
   List[17].Entry_Points[5].operation_type := 'machining';
   List[17].Entry_Points[5].lay_number := -1;
   List[17].Entry_Points[5].operation_side := 'A';
   List[17].Entry_Points[5].part_side := 'A';
   List[17].Entry_Points[6].active := true;
   List[17].Entry_Points[6].previous_trajectory := 'AutoMachining_B';
   List[17].Entry_Points[6].machine_status := 'ready2load';
   List[17].Entry_Points[6].robot_status := 'pallet_out';
   List[17].Entry_Points[6].part_status := 'pallet_in';
   List[17].Entry_Points[6].part_destination := 'flip_table';
   List[17].Entry_Points[6].operation_type := 'machining';
   List[17].Entry_Points[6].lay_number := -1;
   List[17].Entry_Points[6].operation_side := 'A';
   List[17].Entry_Points[6].part_side := 'A';
   List[14].Entry_Points[4].robot_status := 'home';
END_DATA_BLOCK

